// TIA Portal V20 export
FUNCTION_BLOCK "FB_ValveControl"   // FB2, SCL
{ S7_Optimized_Access := 'TRUE' }
// stored: MemoryReserve 100, SetENOAutomatically false
   VAR_INPUT
      bOpen : Bool;
      bClose : Bool;
   END_VAR
   VAR_OUTPUT
      bOpened : Bool;
      bClosed : Bool;
      bFault : Bool;
   END_VAR
BEGIN

   IF #bOpen THEN
       #bOpened := TRUE;
       #bClosed := FALSE;
   END_IF;

   IF #bClose THEN
       #bOpened := FALSE;
       #bClosed := TRUE;
   END_IF;
END_FUNCTION_BLOCK
